FUNCTION fc_DEG : real
VAR_INPUT
		rad : REAL;
END_VAR
VAR
END_VAR

fc_DEG := fc_MODR(57.29577951308232 * RAD, 360.0);

END_FUNCTION

(* stored: Version 1.1.0.1, ProductVersion 3.1.4024.11
   POU fc_DEG: Id {0c0f8bac-048c-4af1-a933-f23836f12c0a}, SpecialFunc None *)
